//---------------------------------------------------------------------------------------------------------------
//
//  HAUD 2024.03.18
//
//  - XTS_TRAINING
//  - example project for setting up transport layer
//  - transport layer members:
//    - CaGroup
//      - access to Group functions
//
//    - Mover
//      - access to MC and CA motion functions
//
//    - Xpu (ProcessingUnit)
//      - access to TcCOM Objects in Environment
//
//    - Transport Control Unit
//      - coordinates members to get XTS in defined states
//
//    - Xts Stations
//      - handshakes with extern control for mover transport
//
//  - global datafields for mrmbers in GVL_XTS namespace
//  - global interface datafields for use in members
//  - structures are assigned by reference for every member
//
//---------------------------------------------------------------------------------------------------------------
// This SOFTWARE is provided as an Exemple by THE PROVIDER "as is" and "with all faults." THE PROVIDER makes no 
// representations or warranties of any kind concerning the safety, suitability, lack of viruses, inaccuracies, 
// typographical errors, or other harmful components of this SOFTWARE. There are inherent dangers in the use of 
// any software, and you are solely responsible for determining whether this SOFTWARE is compatible with your 
// equipment and other software installed on your equipment. You are also solely responsible for the protection 
// of your equipment and backup of your data, and THE PROVIDER will not be liable for any damages you may suffer 
// in connection with using, modifying, or distributing this SOFTWARE.
//---------------------------------------------------------------------------------------------------------------
PROGRAM MAIN
VAR
	bInit 				: BOOL;
  eInit         : E_PROGRESS;

  nStation,
	nMover,
  nMoverSelected			: UINT;

  eTransportState     : E_XTS_TRANSPORT_STATE;
  eTransportResult    : E_PROGRESS;

  eXpuState           : E_XPU_STATE;
  eXpuResult          : E_PROGRESS;
  eXpuCheck           : E_XPU_CHECK;

  eMoverState         : E_MOVER_STATE;
  eMoverResult        : E_PROGRESS;

  sCaGroupState,
  sTransportState,
  sTransportCheck,
  sTransportResult,
  sXpuState,
  sXpuResult,
  sXpuCheck,
  sXpuOpMode,
  sXpuMoverdetectionMode,
  sXpuMoverAssignement,
  sMoverState,
  sMoverResult        : STRING;
END_VAR

//############################################################################
// 	example for init sequence
//############################################################################	
IF NOT bInit
THEN
  CASE eInit
  OF
    E_PROGRESS.PROGRESS_INVALID,
    E_PROGRESS.PROGRESS_DONE:         // clear command interface
      eInit                           := E_PROGRESS.PROGRESS_BUSY;
      GVL_XTS.XpuCtrl.Cmd             := E_XPU_CTRL.XTS_CMD_NULL;

    E_PROGRESS.PROGRESS_BUSY:         // init Xpu, ProcessingUnit, MotorModules
      eInit                           := E_PROGRESS.PROGRESS_PREPARE;
      GVL_XTS.XpuCtrl.Cmd             := E_XPU_CTRL.XTS_CMD_INIT;

    E_PROGRESS.PROGRESS_PREPARE:      // wait for init to be done
      IF (GVL_XTS.XpuState.State      = E_XPU_STATE.XTS_INIT + E_PROGRESS.PROGRESS_DONE)
      THEN
        eInit                         := E_PROGRESS.PROGRESS_STARTUP;
        GVL_XTS.XpuCtrl.Cmd           := E_XPU_CTRL.XTS_IDLE;
      END_IF

    E_PROGRESS.PROGRESS_STARTUP:      // assign mover interfaces
      eInit                           := E_PROGRESS.PROGRESS_CHECK;
      FOR nMover := 1 TO MAX_MOVER
      DO
        GVL_XTS.MoverItf[nMover]      := GVL_XTS.Mover[nMover];
      END_FOR

    E_PROGRESS.PROGRESS_CHECK:        // assign CaGroup interface
      eInit                           := E_PROGRESS.PROGRESS_OCCUPIED;
      GVL_XTS.CaGroupItf              := GVL_XTS.CaGroup;

    E_PROGRESS.PROGRESS_OCCUPIED:     // StartStation for XtsTransportCtrl.Cmd := E_XTS_TRANSPORT_CTRL.CMD_TRANSPORT_START;
      eInit                           := E_PROGRESS.PROGRESS_WORKING;
      // Start Position parameters
      GVL_XTS.StationStart.rPosWait   :=    375.0;
      GVL_XTS.StationStart.rGap       :=    125.0;
      GVL_XTS.StationStart.rVelo      :=   1250.0;
      GVL_XTS.StationStart.rAccDec    :=  12000.0;
      GVL_XTS.StationStart.rJerk      := 400000.0;

    E_PROGRESS.PROGRESS_WORKING:
      GVL_XTS.StationParameter[1].rPosWait            :=   375.0; // absolute modulo position
      GVL_XTS.StationParameter[1].rPosStop[1]         :=   150.0; // relative to rPosWait
      GVL_XTS.StationParameter[1].rReleaseDistance    :=   125.0; // relative to Mover.ActPos

      GVL_XTS.StationParameter[1].rVelo               :=   1250.0;
      GVL_XTS.StationParameter[1].rAccDec             :=  12000.0;
      GVL_XTS.StationParameter[1].rJerk               := 400000.0;


      GVL_XTS.StationParameter[2].rPosWait            :=  1375.0; // absolute modulo position
      GVL_XTS.StationParameter[2].rPosStop[1]         :=   150.0; // relative to rPosWait
      GVL_XTS.StationParameter[2].rReleaseDistance    :=   125.0; // relative to Mover.ActPos

      GVL_XTS.StationParameter[2].rVelo               :=   1250.0;
      GVL_XTS.StationParameter[2].rAccDec             :=  12000.0;
      GVL_XTS.StationParameter[2].rJerk               := 400000.0;

      bInit                                           := TRUE;
      eInit                                           := E_PROGRESS.PROGRESS_DONE;
  END_CASE
END_IF

//############################################################################
// 	XTS Transport Unit
//############################################################################
//  - main control function block for transport layer
//  - requires access to member controls
//    - Xpu
//    - CaGroup
//    - Mover
//    - Station Control
//    - Station LinkedList Interface
//############################################################################
//
// cyclic call
GVL_XTS.XtsTransport();

// main control
GVL_XTS.XtsTransport.Ctrl               REF= GVL_XTS.XtsTransportCtrl;   // main control
GVL_XTS.XtsTransport.State              REF= GVL_XTS.XtsTransportState;  // main state
                                        
// member controls                      
GVL_XTS.XtsTransport.XpuCtrl            REF= GVL_XTS.XpuCtrl;
GVL_XTS.XtsTransport.XpuState           REF= GVL_XTS.XpuState;
GVL_XTS.XtsTransport.XpuInfo            REF= GVL_XTS.XpuInfo;
                                        
GVL_XTS.XtsTransport.GroupItf           :=   GVL_XTS.CaGroupItf;
GVL_XTS.XtsTransport.GroupInfo          REF= GVL_XTS.CaGroupInfo;
                                        
GVL_XTS.XtsTransport.MoverItf           REF= GVL_XTS.MoverItf;
GVL_XTS.XtsTransport.MoverInfo          REF= GVL_XTS.MoverInfo;
                                        
// start position for E_XTS_TRANSPORT_CTRL.CMD_TRANSPORT_START
GVL_XTS.XtsTransport.StationStart       REF= GVL_XTS.StationStart;

// control of stations is required for clearing states and init lists
GVL_XTS.XtsTransport.StationCtrl        REF= GVL_XTS.StationCtrl;

// list interface is required for access to linked list methods
GVL_XTS.XtsTransport.ItfStations        := ADR(GVL_XTS.StationListItf);

// where to start?
GVL_XTS.XtsTransport.StartStationIndex  := 1;
//############################################################################



//############################################################################
// 	XTS Stations
//############################################################################	
FOR nStation := 1 TO MAX_STATION
DO
  GVL_XTS.Station[nStation].StationId   := nStation;

  GVL_XTS.StationListItf[nStation]      := GVL_XTS.StationList[nStation];

  GVL_XTS.Station[nStation].Ctrl        := ADR(GVL_XTS.StationCtrl);
  GVL_XTS.Station[nStation].State       := ADR(GVL_XTS.StationState);

  GVL_XTS.Station[nStation].ItfStations := ADR(GVL_XTS.StationListItf);
  GVL_XTS.Station[nStation].ItfMover    := ADR(GVL_XTS.MoverItf);
  GVL_XTS.Station[nStation].Mover       := ADR(GVL_XTS.AxisRefMover);
  GVL_XTS.Station[nStation].MoverOffset := ADR(GVL_XTS.PositionOffset);


  GVL_XTS.Station[nStation].StationParameter  := ADR(GVL_XTS.StationParameter);

  // cyclic call
  GVL_XTS.Station[nStation].Cycle(); 
END_FOR
//############################################################################



//############################################################################
// 	XPU environment
//############################################################################	
GVL_XTS.Xpu.XpuInstance               := 1;
GVL_XTS.Xpu.Ctrl                      REF= GVL_XTS.XpuCtrl;
GVL_XTS.Xpu.State                     REF= GVL_XTS.XpuState;
GVL_XTS.Xpu.XpuModuleInfoData         REF= GVL_XTS.XpuModules;

GVL_XTS.Xpu.CaGroupOID                :=   GVL_XTS.CaGroup.GroupInfo.CaGroupOID;

// cyclic call
GVL_XTS.Xpu();
GVL_XTS.XpuInfo                       :=   GVL_XTS.Xpu.XpuInfo;
//############################################################################


//############################################################################	
// 	CA-Group Class
//############################################################################	
// assignment
GVL_XTS.CaGroup.AxisRef               REF= GVL_XTS.AxisRefMover;
GVL_XTS.CaGroup.GroupRef              REF= GVL_XTS.CaGroupRef;

// cyclic call
GVL_XTS.CaGroup.InfoCycle(TRUE); // read group status

// InfoData from group
GVL_XTS.CaGroupInfo                   :=   GVL_XTS.CaGroup.GroupInfo;

// Interface of CaGroup
GVL_XTS.CaGroupItf                    :=   GVL_XTS.CaGroup;
//############################################################################


//############################################################################
// Mover Class	
//############################################################################	
FOR nMover := 1 TO MAX_MOVER
DO
  GVL_XTS.Mover[nMover].Ctrl          REF= GVL_XTS.MoverCtrl [nMover];
  GVL_XTS.Mover[nMover].State         REF= GVL_XTS.MoverState[nMover];

  GVL_XTS.Mover[nMover].MoveData      REF= GVL_XTS.MoveData[nMover];
  GVL_XTS.Mover[nMover].GearData      REF= GVL_XTS.GearData[nMover];

  // assignment	
  GVL_XTS.Mover[nMover].Mover         REF= GVL_XTS.AxisRefMover[nMover];  // axis reference to Mover function block
  GVL_XTS.Mover[nMover].LastGap       REF= GVL_XTS.LastGap[nMover];       // reference to last used gap value datafield
  GVL_XTS.Mover[nMover].LastPosition  REF= GVL_XTS.LastPosition[nMover];  // reference to last position datafield
  
  GVL_XTS.Mover[nMover].RailLength    := GVL_XTS.Xpu.RailLength;          // mover needs RailLength, in order to calc absolute position from modulo input
  
  GVL_XTS.Mover[nMover].MoverInfo		  REF= GVL_XTS.MoverInfo[nMover];     // refernence to mover info data (ActPos, SetPos, ...)

  GVL_XTS.MoverItf[nMover]            := GVL_XTS.Mover[nMover];

  // cyclic call
  GVL_XTS.Mover[nMover].Cycle();  // call AXIS_REF()
  GVL_XTS.Mover[nMover]();        // call Ctrl/State
END_FOR


//############################################################################



//############################################################################
// Visualization data	
//############################################################################	
// get enumerations from XPU for visu:
eTransportState                       := f_GetState   (GVL_XTS.XtsTransportState.State);
eTransportResult                      := f_GetProgress(GVL_XTS.XtsTransportState.State);

eXpuState                             := f_GetState   (GVL_XTS.XpuState.State);
eXpuResult                            := f_GetProgress(GVL_XTS.XpuState.State);

eXpuCheck                             := GVL_XTS.XpuState.Check;

// display xpu state and result in visu
// get strings and info
sCaGroupState                         := TO_STRING(GVL_XTS.CaGroupInfo.CaGroupState);

sTransportState                       := TO_STRING(eTransportState);
sTransportCheck                       := TO_STRING(GVL_XTS.XtsTransportState.Check);
sTransportResult                      := TO_STRING(eTransportResult);

sXpuState                             := TO_STRING(eXpuState);
sXpuResult                            := TO_STRING(eXpuResult);
sXpuCheck                             := TO_STRING(eXpuCheck);

sXpuOpMode                            := GVL_XTS.Xpu.OpModeToString();
sXpuMoverdetectionMode                := GVL_XTS.Xpu.IdDetectionModeToString();
sXpuMoverAssignement                  := GVL_XTS.Xpu.MoverPositionAssignementToString();

nMoverSelected                        := SEL((nMoverSelected<1), nMoverSelected, 1);
nMoverSelected                        := SEL((nMoverSelected>MAX_MOVER), nMoverSelected, MAX_MOVER);

eMoverState                           := f_GetState   (GVL_XTS.MoverState[nMoverSelected].State);
eMoverResult                          := f_GetProgress(GVL_XTS.MoverState[nMoverSelected].State);

sMoverState                           := TO_STRING(eMoverState);
sMoverResult                          := TO_STRING(eMoverResult);

END_PROGRAM

(* stored: Version 1.1.0.1, ProductVersion 3.1.4024.12
   POU MAIN: Id {f2e9720a-bda2-4399-8c7d-d9b6e11179c8}, SpecialFunc None *)
